FUNCTION_BLOCK LinkedListNode EXTENDS Disposable IMPLEMENTS I_LinkedListNode
VAR
	internalBuffer : POINTER TO BYTE;
	internalBufferSize : UDINT;
	sourceDataType : T_MAXSTRING;
	previousItem : I_LinkedListNode;
	nextItem : I_LinkedListNode;
END_VAR

METHOD PRIVATE CopyInternalBufferToDestination
VAR_INPUT
	DestinationAddress : PVOID;
END_VAR
memcpy(DestinationAddress,internalBuffer,internalBufferSize);
END_METHOD

METHOD PRIVATE CopySourceToInternalBuffer
VAR_INPUT
	SourceAddress : PVOID;
END_VAR
memcpy(internalBuffer,SourceAddress,internalBufferSize);
END_METHOD

METHOD PRIVATE DeleteInternalBuffer
IF internalBuffer <> 0 THEN
	__DELETE(internalBuffer);
END_IF
END_METHOD

METHOD PUBLIC Equals : BOOL
VAR_INPUT
	Symbol : ANY;
END_VAR
IF NOT IsInternalBufferSameSizeAs(DINT_TO_UDINT(Symbol.diSize)) THEN
	RETURN;
END_IF

Equals := memcmp(Symbol.pValue,internalBuffer,Symbol.diSize) = 0;
END_METHOD

METHOD FB_init : BOOL
VAR_INPUT
	bInitRetains : BOOL; // if TRUE, the retain variables are initialized (warm start / cold start)
	bInCopyCode : BOOL;  // if TRUE, the instance afterwards gets moved into the copy code (online change)
	Source : ANY;
END_VAR
MakeInternalBufferOfSize(DINT_TO_UDINT(Source.diSize));
CopySourceToInternalBuffer(Source.pValue);
END_METHOD

METHOD PUBLIC Get : BOOL;
VAR_INPUT
	Destination : ANY;
END_VAR
Get := GetTo(Destination.pValue,Destination.diSize);
END_METHOD

METHOD PUBLIC GetTo : BOOL;
VAR_INPUT
	Destination : PVOID;
	DestinationSize : UDINT;
END_VAR
IF NOT IsInternalBufferSameSizeAs(DestinationSize) THEN
	RETURN;
END_IF

CopyInternalBufferToDestination(Destination);
GetTo := TRUE;
END_METHOD

METHOD PRIVATE IsInternalBufferSameSizeAs : BOOL
VAR_INPUT
	Size : UDINT;
END_VAR
IF internalBuffer = 0 THEN
	RETURN;
END_IF

IF internalBufferSize <> Size THEN
	RETURN;
END_IF

IsInternalBufferSameSizeAs := TRUE;
END_METHOD

METHOD PRIVATE MakeInternalBufferOfSize
VAR_INPUT
	Size : UDINT;
END_VAR
internalBufferSize := Size;
internalBuffer := __NEW(BYTE, internalBufferSize);
END_METHOD

PROPERTY PUBLIC Next : I_LinkedListNode
GET
Next := nextItem;
END_GET
SET // PUBLIC
nextItem := Next;
END_SET
END_PROPERTY

METHOD PROTECTED OnDispose : BOOL
VAR_INPUT
	CalledExplicitly : BOOL;
END_VAR
DeleteInternalBuffer();
END_METHOD

PROPERTY PUBLIC Previous : I_LinkedListNode
GET
Previous := previousItem;
END_GET
SET // PUBLIC
previousItem := Previous;
END_SET
END_PROPERTY

END_FUNCTION_BLOCK

(* stored: Version 1.1.0.1, ProductVersion 3.1.4024.12
   POU LinkedListNode: Id {145197a1-b0ae-480f-9d2e-3a28cdd2aac5}, SpecialFunc None
   Folder Constructor: Id {4aac0288-157a-4954-9753-704ed032ee83}
   Folder Private: Id {d4cdadcf-db3d-41bf-a95e-c453364157e1}
   Folder Protected: Id {a3faec45-cc9e-4a10-9c3e-289211383e8f}
   Method CopyInternalBufferToDestination: Id {39c976be-1b1c-4ed7-adbe-2b6aff05010c}
   Method CopySourceToInternalBuffer: Id {72a972f5-c332-490c-98b2-fbc57602567b}
   Method DeleteInternalBuffer: Id {0b2f16d0-ea60-47d4-8d2f-cb219d773612}
   Method Equals: Id {691d2391-52f1-4b30-a37b-a11ec95819c6}
   Method FB_init: Id {aa5050e3-7bd5-46f0-bcec-c1565801ee0a}
   Method Get: Id {8f654b85-5f92-4a32-bae0-56ed9c46637f}
   Method GetTo: Id {fa8466a7-5e9f-4b8f-b5d1-da656daf3890}
   Method IsInternalBufferSameSizeAs: Id {4a4ea573-a854-47f7-b261-8c18a0c29be2}
   Method MakeInternalBufferOfSize: Id {07db7bed-34c5-49fe-a6f5-1d4ddef28561}
   Property Next: Id {dedd5018-9eee-4162-a026-681e2d07b1ee}
   Get Get: Id {121648c0-ad4d-4c9f-a728-87b9114faa4f}
   Set Set: Id {0ca43cae-5b30-4615-ad5b-c71b537a241f}
   Method OnDispose: Id {d288edc7-b0a3-4f1b-9d7c-374f4617d931}
   Property Previous: Id {d0b69103-fca9-4fdb-bc73-11778d148ddb}
   Get Get: Id {c9509b01-8bbe-4c3d-975e-21220c339e4d}
   Set Set: Id {48755caa-5e5b-4d2f-b027-f2e48f8cc239} *)
